TYPE EL5032_Data :
STRUCT
	{attribute addProperty Name "FB Inputs Channel 1"}
	FB_InputsChannel_1 : EL5032_FB_InputsChannel;
	{attribute addProperty Name "FB Inputs Channel 2"}
	FB_InputsChannel_2 : EL5032_FB_InputsChannel;
END_STRUCT
END_TYPE

(* stored: Version 1.1.0.1, ProductVersion 3.1.4024.9
   DUT EL5032_Data: Id {876a6053-6ebe-08d6-00a5-c968037ecfa9} *)
